FUNCTION_BLOCK FB_ServiceModule
VAR_INPUT
END_VAR
VAR_OUTPUT
	eCondition : eConditionCheck;
	eState : eHighLevelState;
	
END_VAR
VAR
	fbDistanceSensor : FB_DistanceSensor;
	fbBoxLED : FB_BoxLED;
	fbRGBController : FB_RGBController;
	
	eDistanceSensorLastMessage : eErrorList := eErrorList.NoError;	
END_VAR

fbDistanceSensor();
fbBoxLED();
fbRGBController();

//Condition
IF fbDistanceSensor.eCondition = eConditionCheck.READY THEN
	eCondition := eConditionCheck.READY;
	
	eDistanceSensorLastMessage := eErrorList.NoError;
ELSE
	eCondition := eConditionCheck.INIT;
	
	IF fbDistanceSensor.eErrorID <> eDistanceSensorLastMessage THEN
		eDistanceSensorLastMessage := fbDistanceSensor.eErrorID;
		IF fbDistanceSensor.eErrorID <> eErrorList.NoError THEN
			MainControl.fbErrorHandling.fbErrorBufferDistanceSensor.AddErrorMessage(eErrorMessage := fbDistanceSensor.eErrorID);
		END_IF
	END_IF
	
END_IF
	


//High Level State Machine
CASE MainControl.eMainState OF
	eMainStateMachine.READY :
		setLightMode := eLightMode.Init;
		setLEDColor := eColor.BLUE;
		
		eState := eHighLevelState.OPERATIONAL;
	//
	eMainStateMachine.OPERATIONAL :
		setLightMode := eLightMode.Run;
		setLEDColor := eColor.GREEN;
		MyGVLData.lrDistanceSensorServiceModule := getDistanceSensor;
		
		eState := eHighLevelState.SHUTDOWN;
	//
	eMainStateMachine.SHUTDOWN :
		setLightMode := eLightMode.Shutdown;
		setLEDColor := eColor.RED;
		
		eState := eHighLevelState.READY;
	
	

END_CASE

PROPERTY getDistanceSensor : LREAL
GET
getDistanceSensor := fbDistanceSensor.getDistance;
END_GET
END_PROPERTY

PROPERTY setLEDColor : eColor
SET
fbRGBController.setLEDColor := setLEDColor;
END_SET
END_PROPERTY

PROPERTY setLightMode : eLightMode
SET
fbBoxLED.setLightMode := setLightMode;
END_SET
END_PROPERTY

END_FUNCTION_BLOCK

(* stored: Version 1.1.0.1, ProductVersion 3.1.4024.12
   POU FB_ServiceModule: Id {c2b68249-78b4-4ae5-91f5-9de9a918b256}, SpecialFunc None
   Property getDistanceSensor: Id {2fac17f2-5502-4e29-a71f-8cb1ada492f0}
   Get Get: Id {75a6997a-d806-4312-8a14-3897a8c10414}
   Property setLEDColor: Id {6a7a5b5a-09c5-425d-940e-affb3aa3c15d}
   Set Set: Id {02d5a0ad-12c3-404f-90d8-434fa682923b}
   Property setLightMode: Id {ddaddde0-b0ca-494f-8421-9a4aaeadd879}
   Set Set: Id {005729d2-e110-431a-93b1-2e7c9d259192} *)
